// TIA Portal V17 export
// export: Created 2024-08-26T21:10:48.8091643Z, ExportSetting WithDefaults, DisplayName Totally Integrated Automation Portal, DisplayVersion V17 Update 7, DisplayName TIA Portal Openness, DisplayVersion V17 Update 7, DisplayName TIA Portal Version Control Interface, DisplayVersion V17, DisplayName SINAMICS Startdrive Advanced, DisplayVersion V17 SP2, DisplayName SINAMICS Startdrive G110M, G120, G120C, G120D, G120P, G115D, DisplayVersion V17 SP2, DisplayName SINAMICS Startdrive G130, G150, S120, S150, SINAMICS MV, S210, DisplayVersion V17 SP2, DisplayName STEP 7 Professional, DisplayVersion V17 Update 7, DisplayName STEP 7 Safety, DisplayVersion V17 Update 6, DisplayName WinCC Advanced / Unified PC, DisplayVersion V17 Update 7
FUNCTION "torqueProfinet" : Void   // FC12, LAD
{ S7_Optimized_Access := 'TRUE' }
VERSION : 0.1
// stored: AutoNumber true, IsIECCheckEnabled false, SetENOAutomatically false, UDAEnableTagReadback false
   VAR_TEMP   // added for the SCL form of the ladder/FBD networks
      _w1 : Bool;
   END_VAR
BEGIN

REGION Network 1: HABILITAR HERRAMIENTA
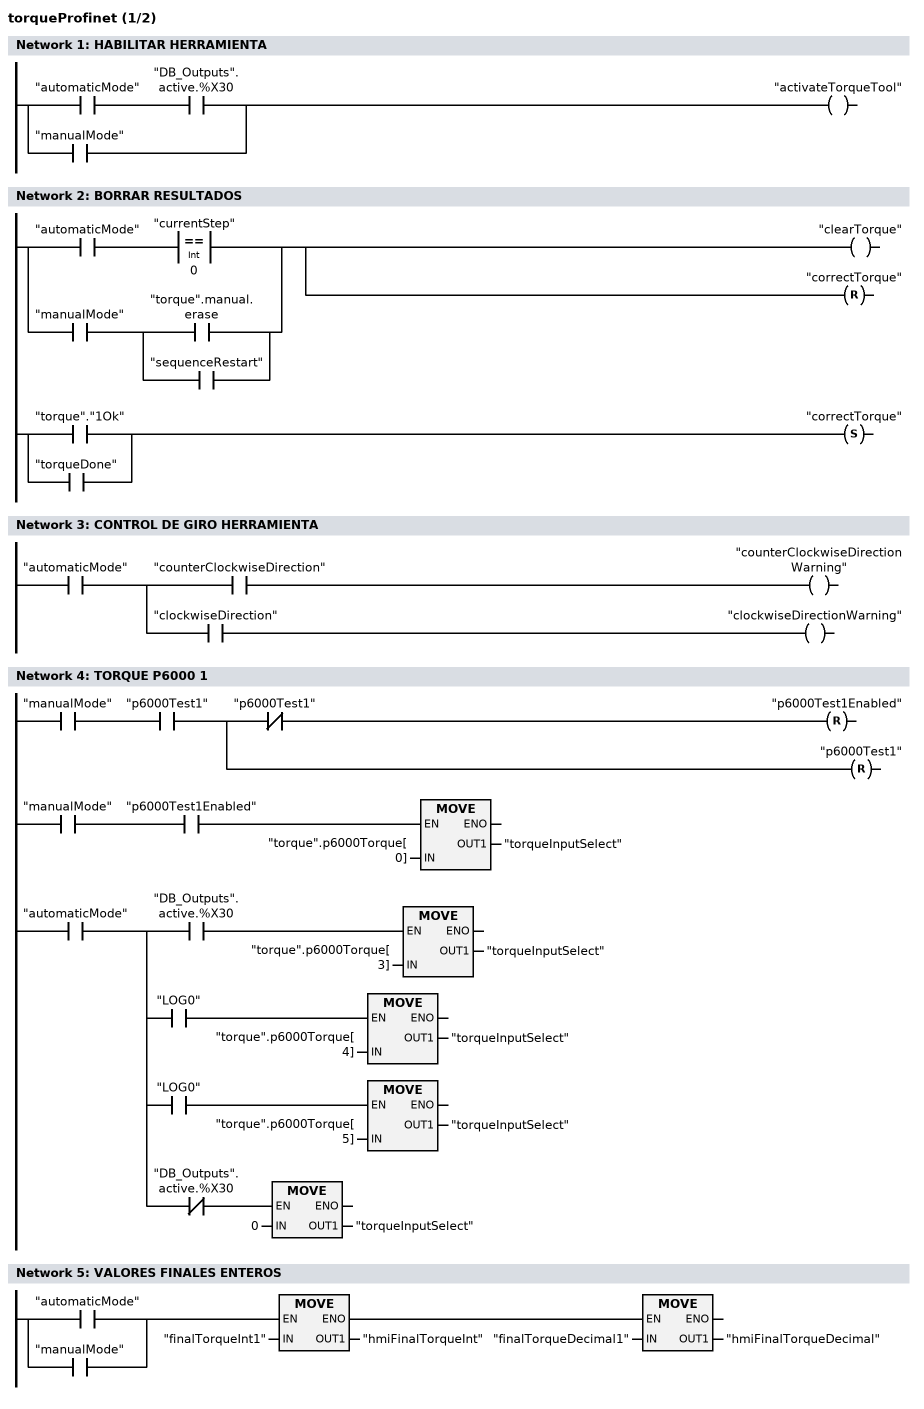
   RUNG wire#powerrail
      Contact( "automaticMode" )
      Contact( "DB_Outputs".active.%X30 )
      wire#w1
      Coil( "activateTorqueTool" )
   END_RUNG
   RUNG wire#powerrail
      Contact( "manualMode" )
   END_RUNG wire#w1
   // the same network as SCL:
   "activateTorqueTool" := ("automaticMode" AND "DB_Outputs".active.%X30) OR "manualMode";
END_REGION

REGION Network 2: BORRAR RESULTADOS
   RUNG wire#powerrail
      Contact( "automaticMode" )
      { S7_Templates := "SrcType := Int" } EQ_Contact(in1 := "currentStep", in2 := 0)
      wire#w1
      Coil( "clearTorque" )
   END_RUNG
   RUNG wire#powerrail
      Contact( "manualMode" )
      wire#w2
      Contact( "torque".manual.erase )
   END_RUNG wire#w1
   RUNG wire#w2
      Contact( "sequenceRestart" )
   END_RUNG wire#w1
   RUNG wire#w1
      R_Coil( "correctTorque" )
   END_RUNG
   RUNG wire#powerrail
      Contact( "torque"."1Ok" )
      wire#w3
      S_Coil( "correctTorque" )
   END_RUNG
   RUNG wire#powerrail
      Contact( "torqueDone" )
   END_RUNG wire#w3
   // the same network as SCL:
   "clearTorque" := ("automaticMode" AND ("currentStep" = 0)) OR ("manualMode" AND ("torque".manual.erase OR "sequenceRestart"));
   IF "clearTorque" THEN "correctTorque" := FALSE; END_IF;
   IF "torque"."1Ok" OR "torqueDone" THEN "correctTorque" := TRUE; END_IF;
END_REGION

REGION Network 3: CONTROL DE GIRO HERRAMIENTA
   RUNG wire#powerrail
      Contact( "automaticMode" )
      wire#w1
      Contact( "counterClockwiseDirection" )
      Coil( "counterClockwiseDirectionWarning" )
   END_RUNG
   RUNG wire#w1
      Contact( "clockwiseDirection" )
      Coil( "clockwiseDirectionWarning" )
   END_RUNG
   // the same network as SCL:
   "counterClockwiseDirectionWarning" := "automaticMode" AND "counterClockwiseDirection";
   "clockwiseDirectionWarning" := "automaticMode" AND "clockwiseDirection";
END_REGION

REGION Network 4: TORQUE P6000 1
   RUNG wire#powerrail
      Contact( "manualMode" )
      Contact( "p6000Test1" )
      wire#w1
      I_Contact( "p6000Test1" )
      R_Coil( "p6000Test1Enabled" )
   END_RUNG
   RUNG wire#w1
      R_Coil( "p6000Test1" )
   END_RUNG
   RUNG wire#powerrail
      Contact( "manualMode" )
      Contact( "p6000Test1Enabled" )
      Move(in := "torque".p6000Torque[0], out1 => "torqueInputSelect")
   END_RUNG
   RUNG wire#powerrail
      Contact( "automaticMode" )
      wire#w2
      Contact( "DB_Outputs".active.%X30 )
      Move(in := "torque".p6000Torque[3], out1 => "torqueInputSelect")
   END_RUNG
   RUNG wire#w2
      Contact( "LOG0" )
      Move(in := "torque".p6000Torque[4], out1 => "torqueInputSelect")
   END_RUNG
   RUNG wire#w2
      Contact( "LOG0" )
      Move(in := "torque".p6000Torque[5], out1 => "torqueInputSelect")
   END_RUNG
   RUNG wire#w2
      I_Contact( "DB_Outputs".active.%X30 )
      Move(in := 0, out1 => "torqueInputSelect")
   END_RUNG
   // the same network as SCL:
   #_w1 := "manualMode" AND "p6000Test1";
   IF #_w1 AND NOT "p6000Test1" THEN "p6000Test1Enabled" := FALSE; END_IF;
   IF #_w1 THEN "p6000Test1" := FALSE; END_IF;
   IF "manualMode" AND "p6000Test1Enabled" THEN "torqueInputSelect" := "torque".p6000Torque[0]; END_IF;
   IF "automaticMode" AND "DB_Outputs".active.%X30 THEN
       "torqueInputSelect" := "torque".p6000Torque[3];
   END_IF;
   IF "automaticMode" AND "LOG0" THEN
       "torqueInputSelect" := "torque".p6000Torque[4];
       "torqueInputSelect" := "torque".p6000Torque[5];
   END_IF;
   IF "automaticMode" AND NOT "DB_Outputs".active.%X30 THEN "torqueInputSelect" := 0; END_IF;
END_REGION

REGION Network 5: VALORES FINALES ENTEROS
   RUNG wire#powerrail
      Contact( "automaticMode" )
      wire#w1
      Move(in := "finalTorqueInt1", out1 => "hmiFinalTorqueInt")
      Move(in := "finalTorqueDecimal1", out1 => "hmiFinalTorqueDecimal")
   END_RUNG
   RUNG wire#powerrail
      Contact( "manualMode" )
   END_RUNG wire#w1
   // the same network as SCL:
   IF "automaticMode" OR "manualMode" THEN
       "hmiFinalTorqueInt" := "finalTorqueInt1";
       "hmiFinalTorqueDecimal" := "finalTorqueDecimal1";
   END_IF;
END_REGION

REGION Network 6
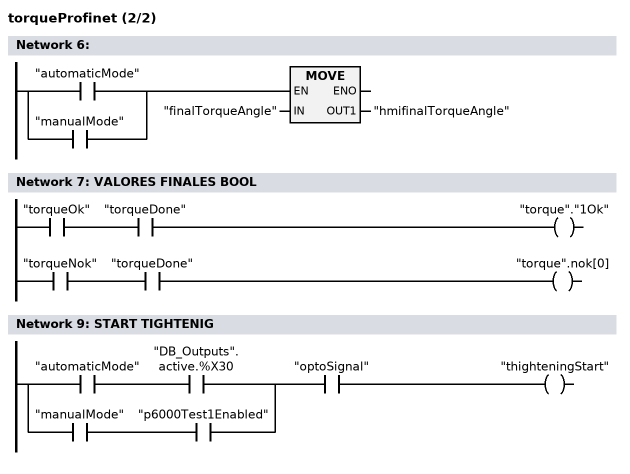
   RUNG wire#powerrail
      Contact( "automaticMode" )
      wire#w1
      Move(in := "finalTorqueAngle", out1 => "hmifinalTorqueAngle")
   END_RUNG
   RUNG wire#powerrail
      Contact( "manualMode" )
   END_RUNG wire#w1
   // the same network as SCL:
   IF "automaticMode" OR "manualMode" THEN "hmifinalTorqueAngle" := "finalTorqueAngle"; END_IF;
END_REGION

REGION Network 7: VALORES FINALES BOOL
   RUNG wire#powerrail
      Contact( "torqueOk" )
      Contact( "torqueDone" )
      Coil( "torque"."1Ok" )
   END_RUNG
   RUNG wire#powerrail
      Contact( "torqueNok" )
      Contact( "torqueDone" )
      Coil( "torque".nok[0] )
   END_RUNG
   // the same network as SCL:
   "torque"."1Ok" := "torqueOk" AND "torqueDone";
   "torque".nok[0] := "torqueNok" AND "torqueDone";
END_REGION

REGION Network 8: TRS
END_REGION

REGION Network 9: START TIGHTENIG
   RUNG wire#powerrail
      Contact( "automaticMode" )
      Contact( "DB_Outputs".active.%X30 )
      wire#w1
      Contact( "optoSignal" )
      Coil( "thighteningStart" )
   END_RUNG
   RUNG wire#powerrail
      Contact( "manualMode" )
      Contact( "p6000Test1Enabled" )
   END_RUNG wire#w1
   // the same network as SCL:
   "thighteningStart" := (("automaticMode" AND "DB_Outputs".active.%X30) OR ("manualMode" AND "p6000Test1Enabled")) AND "optoSignal";
END_REGION
END_FUNCTION
